FUNCTION Convert_UINT_TO_INT : BOOL
VAR_INPUT
	in : UINT;
	out : REFERENCE TO INT;
END_VAR
VAR
	converted : INT;
END_VAR

converted := UINT_TO_INT(in);

IF (INT_TO_UINT(converted) <> in) THEN
	RETURN;
END_IF

out := converted;
Convert_UINT_TO_INT := TRUE;

END_FUNCTION

(* stored: Version 1.1.0.1, ProductVersion 3.1.4024.12
   POU Convert_UINT_TO_INT: Id {d4ea09e6-cd17-4f7e-ab2d-6598fda923b8}, SpecialFunc None *)
